% RSLogix 500 project MM2_BAK032.RSS, saved by version 8.10.00.30 %
PROJECT "UNTITLED"    % processor: Bul.1763 MicroLogix 1100 Series B %

PROGRAM FILES
  LAD 2   5 rungs
  LAD 3 "WATCHDOG"  8 rungs
  LAD 4 "PRODUCT"  8 rungs  % Changes the productcode %
  LAD 5 "REFCTRL"  12 rungs  % Controlling reference measurement %

DATA FILES
  O0 OUTPUT  4 elements
  I1 INPUT  6 elements
  S2 STATUS  66 elements
  B3 BINARY  2 elements
  T4 TIMER  5 elements
  C5 COUNTER  1 elements
  R6 CONTROL  1 elements
  N7 INTEGER  3 elements
  F8 FLOAT  100 elements
  ST9   10 elements
  MG13   1 elements
  RIX15   1 elements
  RI16   1 elements

LADDER 2
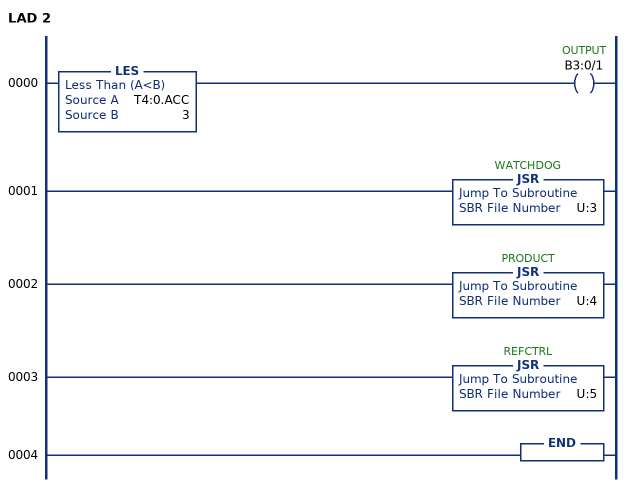
% Rung: 0 %
SOR LES T4:0.ACC 3 OTE B3:0/1 EOR
%   B3:0/1  OUTPUT %
% Rung: 1 %
SOR JSR U:3 EOR
%   U:3  WATCHDOG %
% Rung: 2 %
SOR JSR U:4 EOR
%   U:4  PRODUCT %
% Rung: 3 %
SOR JSR U:5 EOR
%   U:5  REFCTRL %
% Rung: 4 %
SOR END EOR

LADDER 3 "WATCHDOG"
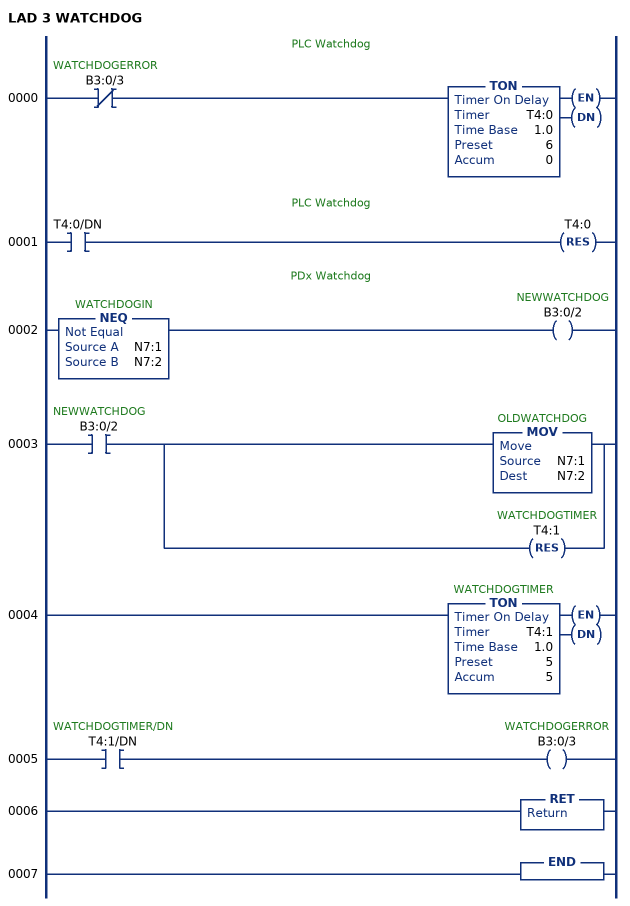
% Rung: 0 %
% PLC Watchdog %
SOR XIO B3:0/3 TON T4:0 1.0 6 0 EOR
%   B3:0/3  WATCHDOGERROR %
% Rung: 1 %
% PLC Watchdog %
SOR XIC T4:0/DN RES T4:0 EOR
% Rung: 2 %
% PDx Watchdog %
SOR NEQ N7:1 N7:2 OTE B3:0/2 EOR
%   N7:1  WATCHDOGIN %
%   N7:2  OLDWATCHDOG %
%   B3:0/2  NEWWATCHDOG %
% Rung: 3 %
SOR XIC B3:0/2 BST MOV N7:1 N7:2 NXB RES T4:1 BND EOR
%   B3:0/2  NEWWATCHDOG %
%   N7:1  WATCHDOGIN %
%   N7:2  OLDWATCHDOG %
%   T4:1  WATCHDOGTIMER %
% Rung: 4 %
SOR TON T4:1 1.0 5 5 EOR
%   T4:1  WATCHDOGTIMER %
% Rung: 5 %
SOR XIC T4:1/DN OTE B3:0/3 EOR
%   T4:1  WATCHDOGTIMER %
%   B3:0/3  WATCHDOGERROR %
% Rung: 6 %
SOR RET EOR
% Rung: 7 %
SOR END EOR

LADDER 4 "PRODUCT"    % Changes the productcode %
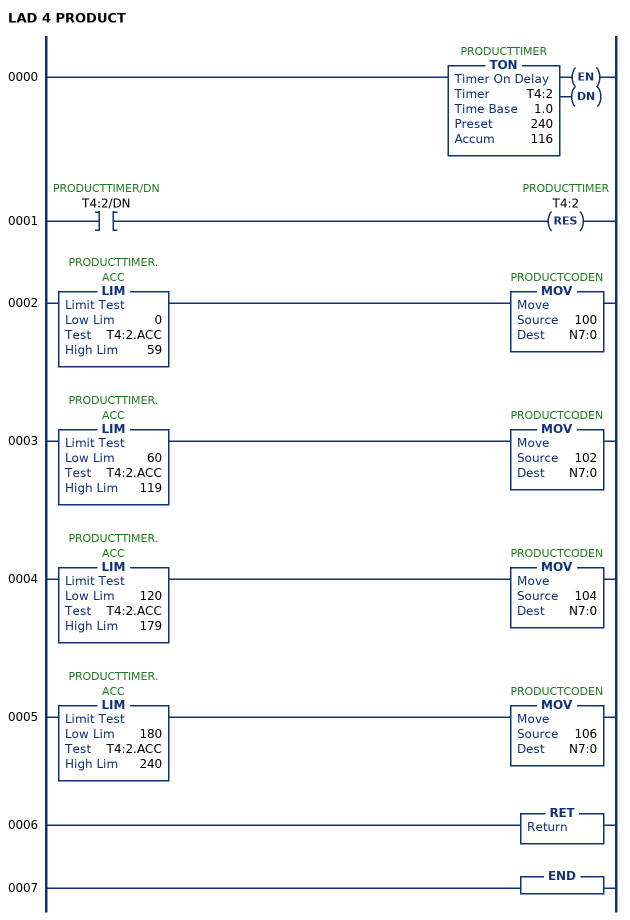
% Rung: 0 %
SOR TON T4:2 1.0 240 116 EOR
%   T4:2  PRODUCTTIMER %
% Rung: 1 %
SOR XIC T4:2/DN RES T4:2 EOR
%   T4:2  PRODUCTTIMER %
% Rung: 2 %
SOR LIM 0 T4:2.ACC 59 MOV 100 N7:0 EOR
%   T4:2  PRODUCTTIMER %
%   N7:0  PRODUCTCODEN %
% Rung: 3 %
SOR LIM 60 T4:2.ACC 119 MOV 102 N7:0 EOR
%   T4:2  PRODUCTTIMER %
%   N7:0  PRODUCTCODEN %
% Rung: 4 %
SOR LIM 120 T4:2.ACC 179 MOV 104 N7:0 EOR
%   T4:2  PRODUCTTIMER %
%   N7:0  PRODUCTCODEN %
% Rung: 5 %
SOR LIM 180 T4:2.ACC 240 MOV 106 N7:0 EOR
%   T4:2  PRODUCTTIMER %
%   N7:0  PRODUCTCODEN %
% Rung: 6 %
SOR RET EOR
% Rung: 7 %
SOR END EOR

LADDER 5 "REFCTRL"    % Controlling reference measurement %
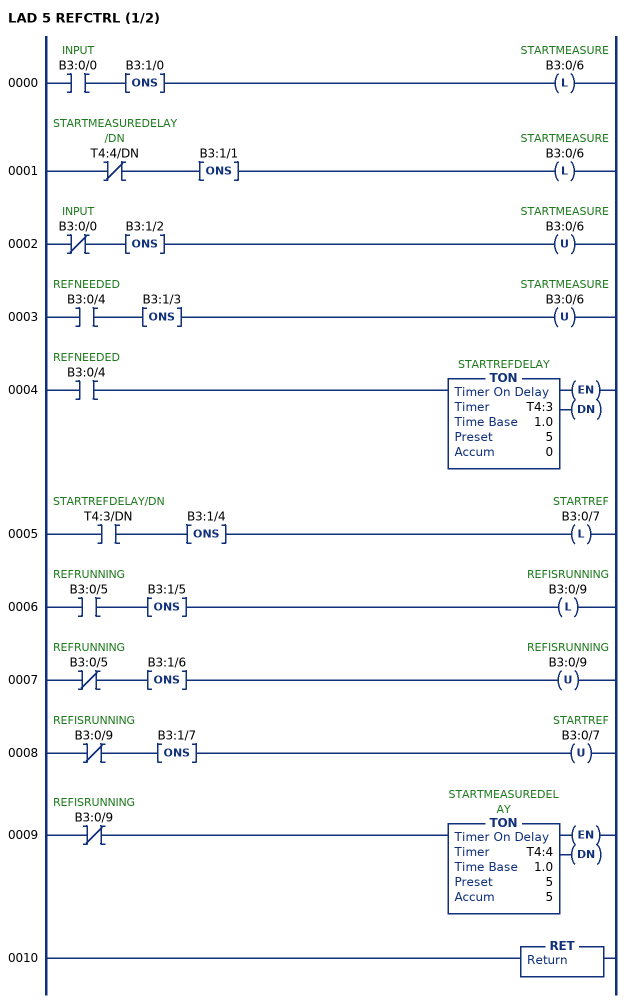
% Rung: 0 %
SOR XIC B3:0/0 ONS B3:1/0 OTL B3:0/6 EOR
%   B3:0/0  INPUT %
%   B3:0/6  STARTMEASURE %
% Rung: 1 %
SOR XIO T4:4/DN ONS B3:1/1 OTL B3:0/6 EOR
%   T4:4  STARTMEASUREDELAY %
%   B3:0/6  STARTMEASURE %
% Rung: 2 %
SOR XIO B3:0/0 ONS B3:1/2 OTU B3:0/6 EOR
%   B3:0/0  INPUT %
%   B3:0/6  STARTMEASURE %
% Rung: 3 %
SOR XIC B3:0/4 ONS B3:1/3 OTU B3:0/6 EOR
%   B3:0/4  REFNEEDED %
%   B3:0/6  STARTMEASURE %
% Rung: 4 %
SOR XIC B3:0/4 TON T4:3 1.0 5 0 EOR
%   B3:0/4  REFNEEDED %
%   T4:3  STARTREFDELAY %
% Rung: 5 %
SOR XIC T4:3/DN ONS B3:1/4 OTL B3:0/7 EOR
%   T4:3  STARTREFDELAY %
%   B3:0/7  STARTREF %
% Rung: 6 %
SOR XIC B3:0/5 ONS B3:1/5 OTL B3:0/9 EOR
%   B3:0/5  REFRUNNING %
%   B3:0/9  REFISRUNNING %
% Rung: 7 %
SOR XIO B3:0/5 ONS B3:1/6 OTU B3:0/9 EOR
%   B3:0/5  REFRUNNING %
%   B3:0/9  REFISRUNNING %
% Rung: 8 %
SOR XIO B3:0/9 ONS B3:1/7 OTU B3:0/7 EOR
%   B3:0/9  REFISRUNNING %
%   B3:0/7  STARTREF %
% Rung: 9 %
SOR XIO B3:0/9 TON T4:4 1.0 5 5 EOR
%   B3:0/9  REFISRUNNING %
%   T4:4  STARTMEASUREDELAY %
% Rung: 10 %
SOR RET EOR

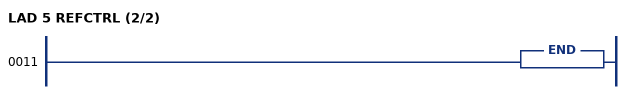
% Rung: 11 %
SOR END EOR

OTHER DOCUMENTED ADDRESSES
  B3:0/8  REFISDONE

DATA TABLE (non-zero values as saved)
DATA B3
% B3:0 % 0X000A 0X00C4
DATA T4
% .PRE .ACC %
% T4:0 % 6 0
% T4:1 % 5 5
% T4:2 % 240 116
% T4:3 % 5 0
% T4:4 % 5 5
DATA C5
% .PRE .ACC %
% C5:0 % 10 0
DATA N7
% N7:0 % 102 730 730
DATA F8
% F8:0 % 65 0 0 0 0
DATA ST9
% ST9:0 % "3"
% ST9:1 % "FDGDGSFB"
% ST9:3 % "GJGJFGN TRFGHNGD"
